(* CoDeSys 2.3 export: DEVICETYPE.EXP *)

(* Data type in ENUM *)
TYPE DeviceType : (System:=1, DiscreteOut, LogicalOut, IODevice, LocalIOManager, NetIOManager, SerialIOManager, LogicSensor,
							DiscreteSensor, ValueSensor, Bin, Transport, Truck, Selector, Batcher, CyclicMixer);
END_TYPE
